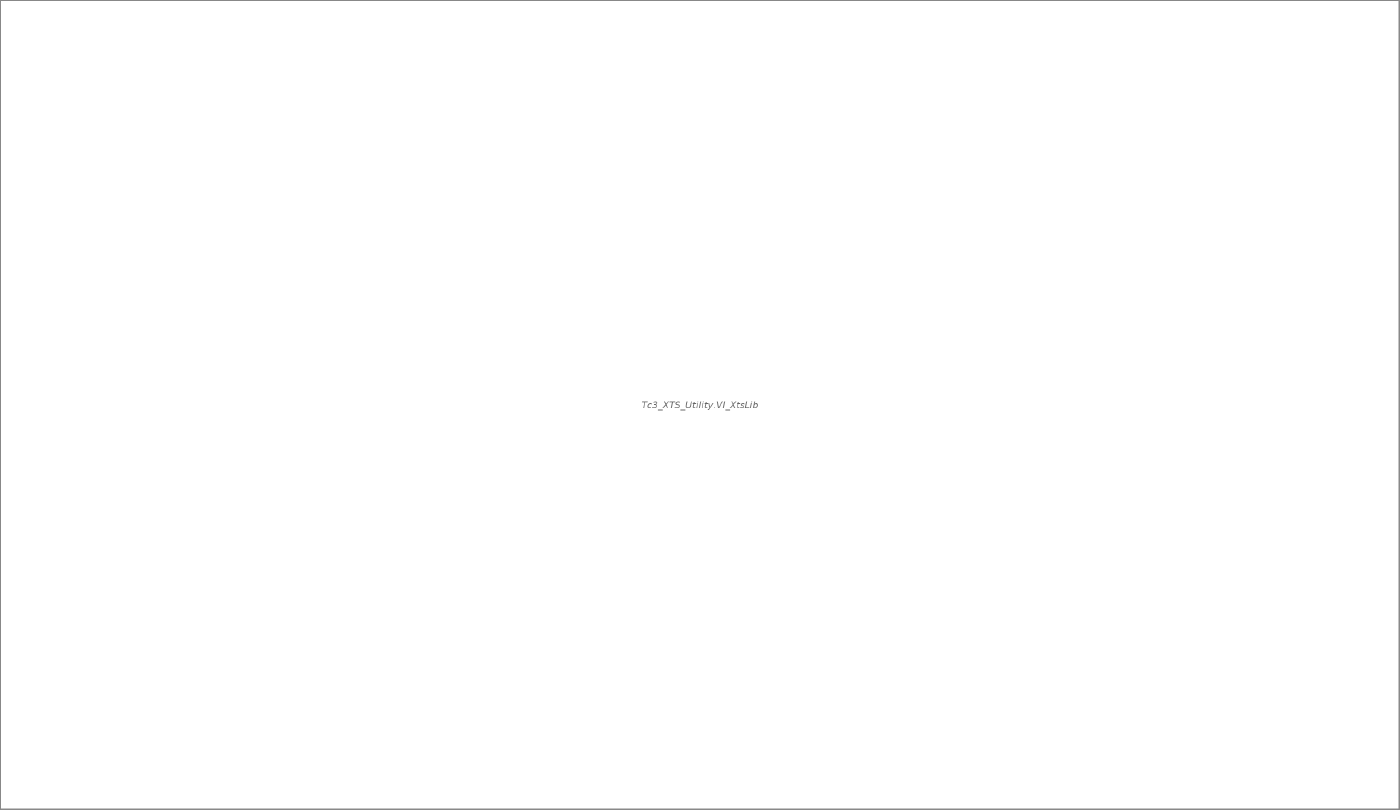
VISUALIZATION PageXtsDiagnostic  // 1520x880
    Frame (0,0 1520x880)
        shows Tc3_XTS_Utility.VI_XtsLib()
END_VISUALIZATION

(* stored: Version 1.1.0.1, ProductVersion 3.1.4024.9
   Visu PageXtsDiagnostic: Id {7132f7cd-50c9-4e46-8517-d59caa0bf868} *)
